FUNCTION_BLOCK OFFSET (* Simple FB with one algorithm *)
  (* Standard: 61499-1; Description: Copyright (c) 2024 HR Agrartechnik GmbH This program and the accompanying materials are made available under the terms of the Eclipse Public License 2.0 which is available at https://www.eclipse.org/legal/epl-2.0/ SPDX-License-Identifier: EPL-2.0 *)
  (* Version 1.0, 2024-10-18, franz *)
  PACKAGE utils::math;
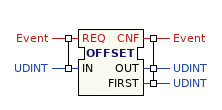
  EVENT_INPUT
    REQ WITH IN; (* Normal Execution Request *)
  END_EVENT
  EVENT_OUTPUT
    CNF WITH OUT, FIRST; (* Execution Confirmation *)
  END_EVENT
  VAR_INPUT
    IN : UDINT; (* Input. First call with a Value &gt;0 will Set FIRST *)
  END_VAR
  VAR_OUTPUT
    OUT : UDINT; (* IN - FIRST *)
    FIRST : UDINT; (* Set at First Call *)
  END_VAR
  ALGORITHM REQ IN ST:
IF (FIRST = 0) THEN
	FIRST := IN;
END_IF;

OUT := IN - FIRST;
  END_ALGORITHM
END_FUNCTION_BLOCK
